(* IEC 61131-3 sources: sps_maggio25/test, 3 files *)

(* ---- testFC.st ---- *)
USING AxUnit;

USING Libreria.Moduli;
USING Libreria.CustomTypes;

NAMESPACE ValveTests

    {Test}
    FUNCTION BasicValveTest

        VAR_TEMP
            testResult : BOOL;
        END_VAR

        BasicValve(cmdOpen := TRUE, ctrlOpen => testResult);
        Assert.Equal(actual := testResult, expected :=TRUE);

    END_FUNCTION

END_NAMESPACE

(* ---- testClass.st ---- *)
USING AxUnit;
USING Libreria.Moduli;
USING Libreria.CustomTypes;

NAMESPACE ValveTests

    {TestFixture}
    CLASS ValveBehaviorTestsCLASS

        VAR PROTECTED
            testInstance : ClassValve;
        END_VAR

        {Test}
        METHOD PUBLIC OpenBehaviorTest

            VAR_TEMP
                result : valveState;
            END_VAR

            testInstance.Open();
            result:= testInstance.GetState();
            Assert.Equal(actual := testInstance.ctrlOpen, expected := TRUE);
            Assert.Equal(actual := result, expected := valveState#Opened);

        END_METHOD

        {Test}
        METHOD PUBLIC CloseBehaviorTest

            VAR_TEMP
                result : valveState;
            END_VAR

            testInstance.Close();
            result:= testInstance.GetState();
            Assert.Equal(actual := testInstance.ctrlOpen, expected := FALSE);
            Assert.Equal(actual := result, expected := valveState#Closed);

        END_METHOD

    END_CLASS

END_NAMESPACE

(* ---- testWrapper.st ---- *)
USING AxUnit;

USING Libreria.Moduli;
USING Libreria.CustomTypes;

NAMESPACE ValveTests

    {TestFixture}
    CLASS ValveBehaviorTestsFB
        VAR
            testInstance : WrapperValve;
        END_VAR

        {Test}
        METHOD PUBLIC WrapperBehaviorTest

            VAR_TEMP
                result : BOOL;
            END_VAR

            testInstance(wCmdOpen := TRUE, wCtrlOpen => result);
            Assert.Equal(actual := result, expected := TRUE);

        END_METHOD

    END_CLASS

END_NAMESPACE
